(* CODESYS project Hugo_Compact.project
   Title: Project.TestTitle
   Author: Project.TestAuthor
   Description: Project.TestDescription
   Version: 3.4.1.0
   Company: Project.TestCompany

Project tree, tasks and I/O mapping:
  CoDeSys_SP_Win_V3 : CoDeSys Control Compact for X86, 3S - Smart Software Solutions GmbH, version 3.4.4.1
    application Application
      task MainTask (cyclic, interval t#25ms, priority 1) calls PLC_PRG
      program PLC_PRG [ST]
      global variables GVL
  CoDeSys_Control_Compact_for_X86 : CoDeSys Control Compact for X86 - With Debugging, 3S - Smart Software Solutions GmbH, version 3.5.0.2
    application Application
      task MainTask (cyclic, interval t#25ms, priority 1) calls PLC_PRG
      program PLC_PRG [ST]
  function GetTitle [ST]
  function GetCompany [ST]
  function GetVersionProperty [ST]
  function GetVersion [ST]
  function GetTextProperty [ST]
  function GetBooleanProperty [ST]
  function GetNumberProperty [ST]
*)

// CoDeSys_SP_Win_V3/Application/GVL
VAR_GLOBAL RETAIN
	dwRetain : DWORD;
END_VAR

// CoDeSys_SP_Win_V3/Application/PLC_PRG
PROGRAM PLC_PRG
VAR
	A: DINT;
	
	MBIT AT %MX1.4 : BOOL;
	M AT %MB1 : BYTE;
	bException : BOOL;
	pFault : POINTER TO DINT;
	tx : BOOL;
	tb : BYTE;
END_VAR

A := A + 100;
dwRetain := dwRetain + 1;

GetTextProperty("");
GetVersionProperty("");

IF bException THEN
	bException := FALSE;
	pFault^:= A;
END_IF
tx := MBIT;
tb := M;

END_PROGRAM

// GetTextProperty
// This function has been automatically generated from the project information.
{attribute 'signature_flag' := '1073741824'}
{attribute 'register_in_runtime'}
FUNCTION GetTextProperty : WSTRING
VAR_INPUT
	stKey: WSTRING;
END_VAR

IF stKey = "Title" THEN
	GetTextProperty := "Project.TestTitle";
ELSIF stKey = "Author" THEN
	GetTextProperty := "Project.TestAuthor";
ELSIF stKey = "Description" THEN
	GetTextProperty := "Project.TestDescription";
ELSIF stKey = "Company" THEN
	GetTextProperty := "Project.TestCompany";
ELSIF stKey = "Project" THEN
	GetTextProperty := "Hugo_Compact";
ELSE
	GetTextProperty := "";
END_IF

END_FUNCTION

// GetVersionProperty
// This function has been automatically generated from the project information.
{attribute 'signature_flag' := '1073741824'}
{attribute 'register_in_runtime'}
FUNCTION GetVersionProperty : VERSION
VAR_INPUT
	stKey: WSTRING;
END_VAR

IF stKey = "Version" THEN
	GetVersionProperty.uiMajor := 3;
	GetVersionProperty.uiMinor := 4;
	GetVersionProperty.uiServicePack := 1;
	GetVersionProperty.uiPatch := 0;
ELSE
	GetVersionProperty.uiMajor := 0;
	GetVersionProperty.uiMinor := 0;
	GetVersionProperty.uiServicePack := 0;
	GetVersionProperty.uiPatch := 0;
END_IF

END_FUNCTION

// CoDeSys_Control_Compact_for_X86/Application/PLC_PRG
PROGRAM PLC_PRG
VAR
	counter: DWORD;
END_VAR

counter := counter + 1;

END_PROGRAM

// GetTitle
// This function has been automatically generated from the project information.
{attribute 'signature_flag' := '1073741824'}
{attribute 'register_in_runtime'}
FUNCTION GetTitle : WSTRING
VAR_INPUT
	
END_VAR

GetTitle := GetTextProperty("Title");

END_FUNCTION

// GetCompany
// This function has been automatically generated from the project information.
{attribute 'signature_flag' := '1073741824'}
{attribute 'register_in_runtime'}
FUNCTION GetCompany : WSTRING
VAR_INPUT
	
END_VAR

GetCompany := GetTextProperty("Company");

END_FUNCTION

// GetVersion
// This function has been automatically generated from the project information.
{attribute 'signature_flag' := '1073741824'}
{attribute 'register_in_runtime'}
FUNCTION GetVersion : VERSION
VAR_INPUT
	
END_VAR

GetVersion := GetVersionProperty("Version");

END_FUNCTION

// GetBooleanProperty
// This function has been automatically generated from the project information.
{attribute 'signature_flag' := '1073741824'}
{attribute 'register_in_runtime'}
FUNCTION GetBooleanProperty : BOOL
VAR_INPUT
	stKey: WSTRING;
END_VAR

GetBooleanProperty := FALSE;

END_FUNCTION

// GetNumberProperty
// This function has been automatically generated from the project information.
{attribute 'signature_flag' := '1073741824'}
{attribute 'register_in_runtime'}
FUNCTION GetNumberProperty : DINT
VAR_INPUT
	stKey: WSTRING;
END_VAR

GetNumberProperty := 0;

END_FUNCTION
